TEXTLIST Stato_WAM
  100 = 'IN ATTESA DI MISSIONE'
  111 = 'CICLO RIPOSO INIT'
  112 = 'CICLO RIPOSO RUN'
  113 = 'WAM CICLO RIPOSO END'
  120 = 'WAM CICLO PALLET INIT'
  121 = 'WAM CICLO PRELIEVO PALLET RUN'
  122 = 'WAM CICLO PRELIEVO PALLET END'
  123 = 'WAM CICLO DEPOSITO PALLET RUN'
  124 = 'WAM CICLO DEPOSITO PALLET END'
  130 = 'WAM CICLO FALDA VUOTI INIT'
  131 = 'WAM CICLO PRELIEVO FALDA VUOTI RUN'
  132 = 'WAM CICLO PRELIEVO FALDA VUOTI END'
  133 = 'WAM CICLO DEPOSITO FALDA VUOTI RUN'
  134 = 'WAM CICLO DEPOSITO FALDA VUOTI END'
  140 = 'WAM CICLO FALDA INIT'
  141 = 'WAM CICLO PRELIEVO FALDA RUN'
  142 = 'WAM CICLO PRELIEVO FALDA END'
  143 = 'WAM CICLO DEPOSITOFALDA RUN'
  144 = 'WAM CICLO DEPOSITO FALDA END'
  150 = 'WAM CICLO PACCO INIT'
  151 = 'WAM CICLO PRELIEVO PACCO RUN'
  152 = 'WAM CICLO PRELIEVO PACCO END'
  153 = 'WAM CICLO DEPOSITO PACCO RUN'
  154 = 'WAM CICLO DEPOSITO PACCO END'
  200 = 'WAMANAGER_CICLO_PRELIEVO_LASTRA_PANCONE_INIT'
  201 = 'CICLO PRELIEVO LASTRA DA PANCONE RUN\n'
  202 = 'WAMANAGER_CICLO_PRELIEVO_LASTRA_DA_PANCONE_END'
  203 = 'WAMANAGER_CICLO_DEPOSITO_LASTRA_PANCONE_INIT'
  204 = 'CICLO DEPOSITO LASTRA SU PANCONE RUN'
  205 = 'WAMANAGER_CICLO_DEPOSITO_LASTRA_SU_PANCONE_END'
  206 = 'WAMANAGER_CICLO_PRELIEVO_LASTRA_DA_CANTILEVER_INIT'
  207 = 'CICLO PRELIEVO LASTRA DA CANTILEVER RUN'
  208 = 'WAMANAGER_CICLO_PRELIEVO_LASTRA_DA_CANTILEVER_END'
  209 = 'WAMANAGER_CICLO_DEPOSITO_LASTRA_SU_CANTILEVER_INIT'
  210 = 'CICLO DEPOSITO LASTRA SU CANTILEVER RUN'
  211 = 'CICLO DEPOSITO LASTRA SU CANTILEVER END'
  212 = 'WAMANAGER_CICLO_POSIZIONAMENTO_SEMPLICE_INIT'
  213 = 'CICLO POSIZIONAMENTO SEMPLICE'
  214 = 'WAMANAGER_CICLO_POSIZONAMENTO_SEMPLICE_END'
  170 = 'WAM CICLO LASTRA INIT'
  171 = 'WAM CICLO PRELIEVO LASTRA RUN'
  172 = 'WAM CICLO PRELIEVO LASTRA END'
  173 = 'WAM CICLO DEPOSITO LASTRA RUN'
  174 = 'WAM CICLO DEPOSITO LASTRA END'
   = ''
END_TEXTLIST

(* stored: Version 1.1.0.1, ProductVersion 3.1.4024.11
   TextList Stato_WAM: Id {156a3abe-45cc-4a7c-bbb6-389120b497f5} *)
